// TwinCAT 3 PLC project Plc
// Title: Template.Essentials
// Company: Template.Essentials
// ProjectVersion: 0.0.0.1
// ProgramVersion: 3.1.4023.0
// libraries:
//   Tc2_Standard, * (Beckhoff Automation GmbH)
//   Tc2_System, * (Beckhoff Automation GmbH)
//   Tc3_Module, * (Beckhoff Automation GmbH)
// project tree:
//   DUTs/ stBools.TcDUT (not stored), stTreeStruct.TcDUT (not stored)
//   / PlcTask.TcTTO (not stored)
//   POUs/ MAIN.TcPOU
// real-time tasks:
//   TASK PlcTask: cycle T#10ms, priority 20, ADS port 350

// ---- POUs/MAIN.TcPOU
PROGRAM MAIN
VAR
	{attribute addProperty Name "<#Hello world#>"}
	Hello_World : stTreeStruct;

END_VAR

END_PROGRAM
